(* CODESYS project CtaAppLeistungsventile_2.0.0.0.library
   Description: Leistungventile Library der CTA
   Version: 2.0.0.0
   Title: CtaAppLeistungventile
   Author: SIS
   DocFormat: reStructuredText
   Placeholder: CtaAppLeistungventile
   LanguageModelAttribute: qualified-access-only
   DefaultNamespace: CtaAppLeistungventile
   CompiledLibraryCompatibilityVersion: CODESYS V3.5 SP16 Patch 3
   Company: CTA

Project tree, tasks and I/O mapping:
  libraries: Standard, 3.5.18.0 (System); CtaSysConfig, 2.0.0.0 (CTA); VisuDialogs, 3.5.16.20 (System); VisuSymbols, 4.5.0.0 (System); CtaVisSymbols, 2.0.0.0 (CTA); CtaAppInfluxLog, 1.0.0.1 (CTA); CtaSysIO, 2.0.0.0 (CTA); CtaSysLeistungventile, 2.0.0.0 (CTA); CtaVisApps, 1.0.0.0 (CTA); CtaVisHelp, 2.0.0.0 (CTA); CtaVisUser, 1.0.0.0 (CTA)
  40 Visualizations/
    CSH/
      PARAMETER/
        visualisation VIS_CSH_PARAMETER
      VISU/
        visualisation VIS_CSH
        visualisation VIS_CSH_QUERY
      ITF_PARAMETER/
        visualisation DIA_CSH_PARAMETER_IO_ITF
      visualisation DIA_CSH
  00000000-0000-0000-0000-000000000000|D:\CoDeSys\LibrariesV3\trunk\Intern\CAA\CAA Template\3.4.0.0 draft\Placeholder.xml
  00000000-0000-0000-0000-000000000000|D:\CoDeSys\LibrariesV3\trunk\Intern\CAA\CAA Template\3.2.0.3 draft\Prefix.pdf
  00000000-0000-0000-0000-000000000000|D:\CoDeSys\LibrariesV3\trunk\Intern\CAA\CAA Template\3.5.2.0 draft\Placeholder.xml
  20 Structs/
    CSV/
      data type scParameter
  50 Images/
  10 Documenation/
    global variables VersionHistory
    global variables readMe
  21 Interface/
    interface ITF_CSH: pro_ITF_CR2, pro_ITF_CR3, pro_ITF_CR4, pro_ITF_CR1, P_tTillCAPStart, P_tTillCAP25, P_tTillCAP100, P_tCR4OffOn
  11 Library Parameter/
  12 Konstanten/
  60 Textlisten/
  13 Globale Variablen/
  text list GlobalTextList
  5ce3da45-db07-42e7-a21c-a00fff4ed8f6|C:\Users\sis\Downloads\dip-switch.svg
  5ce3da45-db07-42e7-a21c-a00fff4ed8f6|C:\Users\sis\Downloads\lightning-bolt-circle.svg
  30 Program Organization Units/
    function block FB_CSH [ST]: metDO_CR4_ON, proDO_CR4_ON, proCR4_ON_ITF, pro_ITF_CR1, pro_ITF_CR2, pro_ITF_CR3, pro_ITF_CR4, actConfig, actTrendLog, P_tCR4OffOn, P_tTillCAP100, P_tTillCAP25, P_tTillCAPStart, metDO_CR1_ON, proDO_CR1_ON, proCR1_ON_ITF, metDO_CR2_ON, proDO_CR2_ON, proCR2_ON_ITF, metDO_CR3_ON, proDO_CR3_ON, proCR3_ON_ITF, FB_INIT
  5ce3da45-db07-42e7-a21c-a00fff4ed8f6|C:\Users\sis\Downloads\sine-wave.svg
  5ce3da45-db07-42e7-a21c-a00fff4ed8f6|C:\Users\sis\Downloads\eye.svg
  5ce3da45-db07-42e7-a21c-a00fff4ed8f6|C:\Users\sis\Downloads\lan.svg
*)

// 20 Structs/CSV/scParameter
TYPE scParameter :
	STRUCT
		tTillCAPStart	:	CtaSysConfig.fbTIME;
		tTillCAP25		:	CtaSysConfig.fbTIME;
		tTillCAP100		:	CtaSysConfig.fbTIME;	
		tCR4OffOn		:	CtaSysConfig.fbTIME;		
	END_STRUCT
END_TYPE

// 10 Documenation/VersionHistory
(* 

.. image:: ../../Images/CTA_Logo.jpg
   :align: right
   :width: 15% 

**Vorlage**   


============ =========== =========== ============================================
**Date**     **Version** **Author**  **Change**
------------ ----------- ----------- --------------------------------------------
04.03.2021   0.0.0.0     SIS         Vorlage erstellt

============ =========== =========== ============================================


*)
VAR_GLOBAL
    stInfo : STRING:= '0.0.0.0, Vorlage, CTA';
END_VAR

// 10 Documenation/readMe
(*

**ReadMe**
 
|	**Empfehlung**
|
|	Bibliothek CtaAppFU zur dämpfung und rampung von Signalen
|	Instanzieren Sie den CtaAppFU.fbFU in ihrem Funktionsbaustein oder POU beispielsweise als fbFUx ( x = Nr. des FU's 
|	Deklarieren Sie die Struktur Variable welche als Parameter und zur ansteuerung dienen wie im Code beispiel.
|  
| *Beispiel* 

+-----------------------+---------------------------------------------------------------------------------------------------------------------------------------------------------------------------------------------------------------------------------------------------------------------------------------------------------------------------------------------------------------------------------------------------------------------------------------+
| Beschreibung          |  Code                                                                                                                                                                                                                                                                                                                                                                                                                                 |
+=======================+=======================================================================================================================================================================================================================================================================================================================================================================================================================================+
| POU oder SmFb         | .. code-block:: codesys                                                                                                                                                                                                                                                                                                                                                                                                               |
|                       |                                                                                                                                                                                                                                                                                                                                                                                                                                       |
|                       |	// Deklaration als VAR im POU oder dem selbsterstellten Funktionsbaustein                                                                                                                                                                                                                                                                                                                                                        	|
|                       |   VAR   																																																				 																																																				|
|						|	    (*Frequenzumformer 1*)																																																		 																																																	|
|						|		fbFU1			: CtaAppFU.fbFU;																																																																																																|
|			 			|	END_VAR                                                                                                                                                                                                                                                                                                                                                                                                                          	|
+-----------------------+---------------------------------------------------------------------------------------------------------------------------------------------------------------------------------------------------------------------------------------------------------------------------------------------------------------------------------------------------------------------------------------------------------------------------------------+
| Code für Init         | .. code-block:: codesys                                                                                                                                                                                                                                                                                                                                                                                                               |
|                       |   																																																					 																																																				|
|			 			|	// Kopieren des nachfolgenden Codes in eine Action zur Initialisierung der Parameter. Zum Beispiel actConfig.																																																				 																										|
|                       |	{region "Parameter Temperaturfühler 1"}                                                                                                                                                                                                                                                                                                                                                                                             |
|			 			|		(*Basis*)                                                                                                                                                                                                                                                                                                                                                                                                                       |
|						|		fbFU1.scParameter.scModBus.fbxMbErrorAsWarning					(_WertInit := FALSE																	 	 		);     //P1 Parameter zur behandlung eines ModBus Fehlers als Warnung.																																															|
|						|	{endregion}                                                                                                                                                      																																																																    | 
|						|																																																																																																										|
+-----------------------+---------------------------------------------------------------------------------------------------------------------------------------------------------------------------------------------------------------------------------------------------------------------------------------------------------------------------------------------------------------------------------------------------------------------------------------+
*)                                                                                                                                                                                                                                                                                                                                                                                                                                                               
VAR_GLOBAL
	xReadMeDone              :   BOOL; 
END_VAR

// 30 Program Organization Units/FB_CSH
FUNCTION_BLOCK FB_CSH EXTENDS CtaSysLeistungventile.FB_LEISTUNGSVENTILE_BASE IMPLEMENTS ITF_CSH
VAR_INPUT
END_VAR
VAR_OUTPUT
END_VAR
VAR	
	// TON
	TON_CAPStart		:	Standard.TON;
	TON_CR4On			:	Standard.TON;	
	TON_CR4Off			:	Standard.TON;
	TON_CAPUp			:	Standard.TON;
	TON_CAPDown			:	Standard.TON;

	// CASE VARIABLEN
	iStepCAPUP			:	INT	:= 1;
	iStepCAPDown		:	INT	:= 1;
	
	// FLANKEN
	pUp					:	Standard.R_TRIG;
	pDown				:	Standard.R_TRIG;
	
	// ZU UND WEGSCHALTZEITEN
	tPerCAPUp			:	TIME;
	tPerCAPDown			:	TIME;
	
	(* Trend Log *)
	fbTrendxCr1			:	CtaAppInfluxLog.FB_LOG_NODE_BOOL;
	fbTrendxCr2			:	CtaAppInfluxLog.FB_LOG_NODE_BOOL;
	fbTrendxCr3			:	CtaAppInfluxLog.FB_LOG_NODE_BOOL;
	fbTrendxCr4			:	CtaAppInfluxLog.FB_LOG_NODE_BOOL;
	fbTrendiCap			:	CtaAppInfluxLog.FB_LOG_NODE_INT;
	
	// Var
	
	xHasBeenReleasedFirst	:	BOOL;
	(* Config *)
	fbConfigFile		:	CtaSysConfig.fbConfigFile;	
	scParameter			:	scParameter;
END_VAR

actConfig();

tPerCAPUp 	:=	scParameter.tTillCAP100.proValue 	/ 4;
tPerCAPDown :=	scParameter.tTillCAP25.proValue		/ 4;	

// Generation of pulses for CR4
TON_CR4On(In := NOT TON_CR4Off.Q ,PT := scParameter.tCR4OffOn.proValue);
TON_CR4Off(In := TON_CR4On.Q ,PT := scParameter.tCR4OffOn.proValue);

IF proRelease THEN
	
	iStepCAPDown := 1;
	
	TON_CAPStart(In := proRelease ,PT := scParameter.tTillCAPStart.proValue);
	
	xHasBeenReleasedFirst := TRUE;
	
	IF TON_CAPStart.Q THEN
		IF scParameter.tTillCAP100.proValue <= T#0S THEN	
			xCR1	:= FALSE;
			xCR2	:= FALSE;
			xCR3 	:= FALSE;
			xCR4	:= TON_CR4On.Q;
			
			xAcknowledge := FALSE;	
		ELSE
			
			xAcknowledge := TRUE;
			
			pUp(CLK := TON_CAPUp.Q);
		
			IF pUp.Q AND iStepCAPUP >= 1 AND iStepCAPUP < 4 THEN
				iStepCAPUP := iStepCAPUP + 1;
			END_IF
	
			CASE iStepCAPUP OF				
			
				1:	// 25%
					xCR1 := FALSE;
					xCR2 := FALSE;
					xCR3 := TRUE;
					xCR4 :=  TON_CR4On.Q;
					iCAP := 25;
			
				2:	// 50%
					xCR1 := FALSE;
					xCR2 := TRUE;
					xCR3 := FALSE;
					xCR4 := TON_CR4On.Q;
					iCAP := 50;
					
				3:	// 75%
					xCR1 := TRUE;
					xCR2 := FALSE;
					xCR3 := FALSE;
					xCR4 := TON_CR4On.Q;
					iCAP := 75;
					
				4:	// 100%
					xCR1 := FALSE;
					xCR2 := FALSE;
					xCR3 := FALSE;
					xCR4 := TON_CR4On.Q;
					iCAP := 100;			
			END_CASE
			
			TON_CAPUp(	IN := NOT TON_CAPUp.Q AND iStepCAPUP < 4,
							PT := tPerCAPUp);
			
		END_IF			
	
	ELSE
		xCR1 := FALSE;
		xCR2 := FALSE;
		xCR3 := TRUE;
		xCR4 := FALSE;
		
		xAcknowledge := FALSE;
	END_IF
ELSE
	IF xHasBeenReleasedFirst THEN
		
		iStepCAPUP := 1;
		
		pDown(CLK := TON_CAPDown.Q);
	
		IF pDown.Q AND iStepCAPDown >= 1 AND iStepCAPDown < 4 THEN
			iStepCAPDown := iStepCAPDown + 1;
		END_IF		
		
		CASE iStepCAPDown OF		
			
				1: // 75%
					xCR1 := TRUE;
					xCR2 := FALSE;
					xCR3 := FALSE;
					xCR4 := TON_CR4On.Q;
					iCAP := 75;
					xAcknowledge := TRUE;
				2: // 50%
					xCR1 := FALSE;
					xCR2 := TRUE;
					xCR3 := FALSE;
					xCR4 := TON_CR4On.Q;
					iCAP := 50;
					xAcknowledge := TRUE;
				3: // 25%
					xCR1 := FALSE;
					xCR2 := FALSE;
					xCR3 := TRUE;
					xCR4 :=  TON_CR4On.Q;
					iCAP := 25;
					xAcknowledge := TRUE;
				4: // Stop
					xCR1 := FALSE;
					xCR2 := FALSE;
					xCR3 := TRUE;
					xCR4 := FALSE;	
					iCAP := 25;
					xAcknowledge := FALSE;	
					xHasBeenReleasedFirst := FALSE;
		END_CASE	
		
		TON_CAPDown(	IN := NOT TON_CAPDown.Q AND iStepCAPDown < 4,
						PT := tPerCAPDown);
	END_IF	
END_IF

IF __QUERYINTERFACE(ITF_BMK,ITF_BMK) THEN
	actTrendlog();
END_IF

METHOD metDO_CR4_ON : BOOL
VAR_INPUT
    ITF_IN		:	CtaSysIO.ITF_IO;
END_VAR
VAR	
	ITF_DO		:	CtaSysIO.ITF_DO;
END_VAR
IF ITF_IN <> 0 THEN	
	ITF_xCR4_ON := ITF_IN;
	IF __QUERYINTERFACE(ITF_xCR4_ON,ITF_DO) THEN		
		ITF_DO.proValue := xCR4;
	END_IF	
ELSE
	metDO_CR4_ON := xCR4;
END_IF
END_METHOD

PROPERTY proDO_CR4_ON : BOOL
GET
proDO_CR4_ON := xCR4;
END_GET
END_PROPERTY

PROPERTY proCR4_ON_ITF : CtaSysIO.ITF_IO
GET
proCR4_ON_ITF := ITF_xCR4_ON;
END_GET
END_PROPERTY

PROPERTY pro_ITF_CR1 : CtaSysIO.ITF_IO
GET
pro_ITF_CR1 := ITF_xCR1_ON;
END_GET
END_PROPERTY

PROPERTY pro_ITF_CR2 : CtaSysIO.ITF_IO
GET
pro_ITF_CR2 := ITF_xCR2_ON;
END_GET
END_PROPERTY

PROPERTY pro_ITF_CR3 : CtaSysIO.ITF_IO
GET
pro_ITF_CR3 := ITF_xCR3_ON;
END_GET
END_PROPERTY

PROPERTY pro_ITF_CR4 : CtaSysIO.ITF_IO
GET
pro_ITF_CR4 := ITF_xCR4_ON;
END_GET
END_PROPERTY

ACTION actConfig:
fbConfigFile();

	scParameter.tTillCAPStart	(_usiParaNr := 1,	itfConfigFb := fbConfigFile);
	scParameter.tTillCAP25		(_usiParaNr := 2,	itfConfigFb := fbConfigFile);
	scParameter.tTillCAP100		(_usiParaNr := 3,	itfConfigFb := fbConfigFile);
	scParameter.tCR4OffOn		(_usiParaNr := 4,	itfConfigFb := fbConfigFile);
END_ACTION

ACTION actTrendLog:
(* CR1 *)
fbTrendxCr1.ENABLE		:= TRUE;
fbTrendxCr1.KEY			:= CONCAT(ITF_BMK.proGetObjectId,'_xCR1');
fbTrendxCr1.SET_VALUE	:= xCR1;

(* CR2 *)
fbTrendxCr2.ENABLE		:= TRUE;
fbTrendxCr2.KEY			:= CONCAT(ITF_BMK.proGetObjectId,'_xCR2');
fbTrendxCr2.SET_VALUE	:= xCR2;

(* CR3 *)
fbTrendxCr3.ENABLE		:= TRUE;
fbTrendxCr3.KEY			:= CONCAT(ITF_BMK.proGetObjectId,'_xCR3');
fbTrendxCr3.SET_VALUE	:= xCR3;

(* CR4 *)
fbTrendxCr4.ENABLE		:= TRUE;
fbTrendxCr4.KEY			:= CONCAT(ITF_BMK.proGetObjectId,'_xCR4');
fbTrendxCr4.SET_VALUE	:= xCR4;

(* actCAP *)
fbTrendiCap.ENABLE		:= TRUE;
fbTrendiCap.KEY			:= CONCAT(ITF_BMK.proGetObjectId,'_iCAP');
fbTrendiCap.SET_VALUE	:= iCAP;
END_ACTION

PROPERTY P_tCR4OffOn : CtaSysConfig.ITF_DATATYPE
GET
P_tCR4OffOn := scParameter.tCR4OffOn;
END_GET
END_PROPERTY

PROPERTY P_tTillCAP100 : CtaSysConfig.ITF_DATATYPE
GET
P_tTillCAP100 := scParameter.tTillCAP100;
END_GET
END_PROPERTY

PROPERTY P_tTillCAP25 : CtaSysConfig.ITF_DATATYPE
GET
P_tTillCAP25 := scParameter.tTillCAP25;
END_GET
END_PROPERTY

PROPERTY P_tTillCAPStart : CtaSysConfig.ITF_DATATYPE
GET
P_tTillCAPStart := scParameter.tTillCAPStart;
END_GET
END_PROPERTY

METHOD metDO_CR1_ON : BOOL
VAR_INPUT
    ITF_IN		:	CtaSysIO.ITF_IO;
END_VAR
VAR	
	ITF_DO		:	CtaSysIO.ITF_DO;
END_VAR
IF ITF_IN <> 0 THEN	
	ITF_xCR1_ON := ITF_IN;
	IF __QUERYINTERFACE(ITF_xCR1_ON,ITF_DO) THEN		
		ITF_DO.proValue := xCR1;
	END_IF	
ELSE
	metDO_CR1_ON := xCR1;
END_IF
END_METHOD

PROPERTY proDO_CR1_ON : BOOL
GET
proDO_CR1_ON := xCR1;
END_GET
END_PROPERTY

PROPERTY proCR1_ON_ITF : CtaSysIO.ITF_IO
GET
proCR1_ON_ITF := ITF_xCR1_ON;
END_GET
END_PROPERTY

METHOD metDO_CR2_ON : BOOL
VAR_INPUT
    ITF_IN		:	CtaSysIO.ITF_IO;
END_VAR
VAR	
	ITF_DO		:	CtaSysIO.ITF_DO;
END_VAR
IF ITF_IN <> 0 THEN	
	ITF_xCR2_ON := ITF_IN;
	IF __QUERYINTERFACE(ITF_xCR2_ON,ITF_DO) THEN		
		ITF_DO.proValue := xCR2;
	END_IF	
ELSE
	metDO_CR2_ON := xCR2;
END_IF
END_METHOD

PROPERTY proDO_CR2_ON : BOOL
GET
proDO_CR2_ON := xCR2;
END_GET
END_PROPERTY

PROPERTY proCR2_ON_ITF : CtaSysIO.ITF_IO
GET
proCR2_ON_ITF := ITF_xCR2_ON;
END_GET
END_PROPERTY

METHOD metDO_CR3_ON : BOOL
VAR_INPUT
    ITF_IN		:	CtaSysIO.ITF_IO;
END_VAR
VAR	
	ITF_DO		:	CtaSysIO.ITF_DO;
END_VAR
IF ITF_IN <> 0 THEN	
	ITF_xCR3_ON := ITF_IN;
	IF __QUERYINTERFACE(ITF_xCR3_ON,ITF_DO) THEN		
		ITF_DO.proValue := xCR3;
	END_IF	
ELSE
	metDO_CR3_ON := xCR3;
END_IF
END_METHOD

PROPERTY proDO_CR3_ON : BOOL
GET
proDO_CR3_ON := xCR3;
END_GET
END_PROPERTY

PROPERTY proCR3_ON_ITF : CtaSysIO.ITF_IO
GET
proCR3_ON_ITF := ITF_xCR3_ON;
END_GET
END_PROPERTY

//FB_Init ist immer implizit verfügbar und wird primär für die Initialisierung verwendet.
//Der Rückgabewert wird nicht ausgewertet. Für gezielte Einflussnahme können Sie
//die Methoden explizit deklarieren und darin mit dem Standard-Initialisierungscode 
//zusätzlichen Code bereitstellen. Sie können den Rückgabewert auswerten.
METHOD FB_Init: BOOL
VAR_INPUT    
bInitRetains: BOOL; // TRUE: Die Retain-Variablen werden initialisiert (Reset warm / Reset kalt)    
bInCopyCode: BOOL;  // TRUE: Die Instanz wird danach in den Kopiercode kopiert (Online-Change)
END_VAR
SUPER^.stVisuDiaName := 'CtaAppLeistungventile.DIA_CSH';
END_METHOD

END_FUNCTION_BLOCK

// 21 Interface/ITF_CSH
INTERFACE ITF_CSH EXTENDS CtaSysLeistungventile.ITF_LEISTUNGSVENTILE_BASE

PROPERTY pro_ITF_CR2 : CtaSysIO.ITF_IO
GET
END_GET
END_PROPERTY

PROPERTY pro_ITF_CR3 : CtaSysIO.ITF_IO
GET
END_GET
END_PROPERTY

PROPERTY pro_ITF_CR4 : CtaSysIO.ITF_IO
GET
END_GET
END_PROPERTY

PROPERTY pro_ITF_CR1 : CtaSysIO.ITF_IO
GET
END_GET
END_PROPERTY

PROPERTY P_tTillCAPStart : CtaSysConfig.ITF_DATATYPE
GET
END_GET
END_PROPERTY

PROPERTY P_tTillCAP25 : CtaSysConfig.ITF_DATATYPE
GET
END_GET
END_PROPERTY

PROPERTY P_tTillCAP100 : CtaSysConfig.ITF_DATATYPE
GET
END_GET
END_PROPERTY

PROPERTY P_tCR4OffOn : CtaSysConfig.ITF_DATATYPE
GET
END_GET
END_PROPERTY

END_INTERFACE

// 40 Visualizations/CSH/PARAMETER/VIS_CSH_PARAMETER
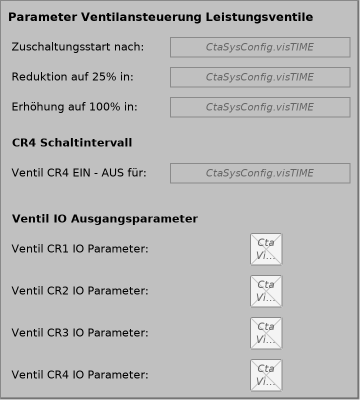
VISUALIZATION VIS_CSH_PARAMETER  // 360x400
VAR_INPUT	
	ITF_CSH_IN				:	ITF_CSH;
	ITF_CR1_IN				:	CtaSysIO.ITF_IO;
	ITF_CR2_IN				:	CtaSysIO.ITF_IO;
	ITF_CR3_IN				:	CtaSysIO.ITF_IO;
	ITF_CR4_IN				:	CtaSysIO.ITF_IO;	
END_VAR
    RoundedRectangle (0,0 358x398)
    Frame (170,37 180x20)
        shows CtaSysConfig.visTIME(visfbTIMEIn := ITF_CSH_IN.P_tTillCAPStart)
    Frame (170,67 180x20)
        shows CtaSysConfig.visTIME(visfbTIMEIn := ITF_CSH_IN.P_tTillCAP25)
    Frame (170,97 180x20)
        shows CtaSysConfig.visTIME(visfbTIMEIn := ITF_CSH_IN.P_tTillCAP100)
    Frame (170,163 180x20)
        shows CtaSysConfig.visTIME(visfbTIMEIn := ITF_CSH_IN.P_tCR4OffOn)
    Label (5,37 150x20), "Zuschaltungsstart nach:"
    Label (5,67 150x20), "Reduktion auf 25% in:"
    Label (5,97 150x20), "Erhöhung auf 100% in:"
    Label (5,163 150x20), "Ventil CR4 EIN - AUS für:"
    Label (5,233 150x32), "Ventil CR1 IO Parameter:", invisible if: ITF_CR1_IN = 0
    Label (5,275 150x32), "Ventil CR2 IO Parameter:", invisible if: ITF_CR2_IN = 0
    Label (5,317 150x32), "Ventil CR3 IO Parameter:", invisible if: ITF_CR3_IN = 0
    Label (5,359 150x32), "Ventil CR4 IO Parameter:", invisible if: ITF_CR4_IN = 0
    Image (250,233 32x32), invisible if: ITF_CR1_IN = 0, input disabled if: ITF_CR1_IN = 0, image: CtaVisSymbols.ImagePool.build
        OnMouseClick:  Dialog=DIA_CSH_PARAMETER_IO_ITF, Parameters={ITF_IO_IN: ITF_CR1_IN}, OpenModal=True, OpenCentered=True
    Image (250,275 32x32), invisible if: ITF_CR2_IN = 0, input disabled if: ITF_CR2_IN = 0, image: CtaVisSymbols.ImagePool.build
        OnMouseClick:  Dialog=DIA_CSH_PARAMETER_IO_ITF, Parameters={ITF_IO_IN: ITF_CR2_IN}, OpenModal=True, OpenCentered=True
    Image (250,317 32x32), invisible if: ITF_CR3_IN = 0, input disabled if: ITF_CR3_IN = 0, image: CtaVisSymbols.ImagePool.build
        OnMouseClick:  Dialog=DIA_CSH_PARAMETER_IO_ITF, Parameters={ITF_IO_IN: ITF_CR3_IN}, OpenModal=True, OpenCentered=True
    Image (250,359 32x32), invisible if: ITF_CR4_IN = 0, input disabled if: ITF_CR4_IN = 0, image: CtaVisSymbols.ImagePool.build
        OnMouseClick:  Dialog=DIA_CSH_PARAMETER_IO_ITF, Parameters={ITF_IO_IN: ITF_CR4_IN}, OpenModal=True, OpenCentered=True
    Label (5,133 250x20), "CR4 Schaltintervall"
    Label (5,7 350x20), "Parameter Ventilansteuerung Leistungsventile"
    Label (5,209 250x20), "Ventil IO Ausgangsparameter", invisible if: ITF_CR1_IN = 0 AND ITF_CR2_IN = 0 AND ITF_CR3_IN = 0 AND ITF_CR4_IN = 0
END_VISUALIZATION

// 40 Visualizations/CSH/VISU/VIS_CSH
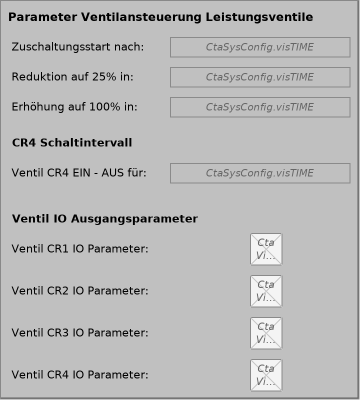
VISUALIZATION VIS_CSH  // 360x400
VAR_INPUT
	ITF_CSH_IN	:	ITF_CSH;
END_VAR
    Frame (0,0 360x400), invisible if: NOT __QUERYINTERFACE(ITF_CSH_IN,ITF_CSH_IN)
        shows VIS_CSH_QUERY(ITF_CSH_IN := ITF_CSH_IN)
END_VISUALIZATION

// 40 Visualizations/CSH/VISU/VIS_CSH_QUERY
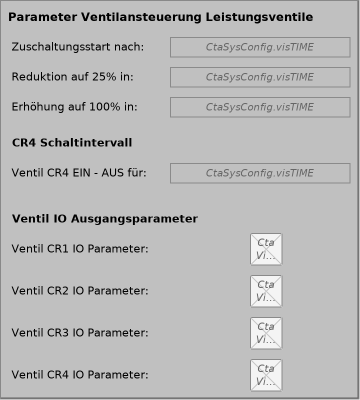
VISUALIZATION VIS_CSH_QUERY  // 360x400
VAR_INPUT
	ITF_CSH_IN	:	ITF_CSH;
END_VAR
    Frame (0,0 360x400)
        shows VIS_CSH_PARAMETER(ITF_CSH_IN := ITF_CSH_IN, ITF_CR1_IN := ITF_CSH_IN.pro_ITF_CR1, ITF_CR2_IN := ITF_CSH_IN.pro_ITF_CR2, ITF_CR3_IN := ITF_CSH_IN.pro_ITF_CR3, ITF_CR4_IN := ITF_CSH_IN.pro_ITF_CR4)
END_VISUALIZATION

// 40 Visualizations/CSH/ITF_PARAMETER/DIA_CSH_PARAMETER_IO_ITF
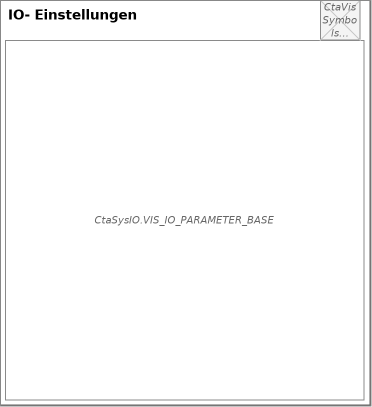
VISUALIZATION DIA_CSH_PARAMETER_IO_ITF  // 372x407
VAR_INPUT
    ITF_IO_IN    :   CtaSysIO.ITF_IO;	
END_VAR
    RoundedRectangle (0,0 370x405)
    Frame (5,40 359x360)
        shows CtaSysIO.VIS_IO_PARAMETER_BASE(ITF_IO_IN := ITF_IO_IN)
        shows VIS_ANTRIEB_PARAMETER_IO1(ITF_ANTRIEBIN := ITF_ANTRIEBIN)
        shows VIS_ANTRIEB_PARAMETER_IO2(ITF_ANTRIEBIN := ITF_ANTRIEBIN)
        shows VIS_ANTRIEB_PARAMETER_IO3(ITF_ANTRIEBIN := ITF_ANTRIEBIN)
    Image (320,0 40x40), image: CtaVisSymbols.ImagePool.close_solo_black
        OnMouseClick:  Dialog=DIA_CSH_PARAMETER_IO_ITF, Result=None, NumpadKeypadSet=True
    Label (5,5 150x20), "IO- Einstellungen"
END_VISUALIZATION

// 40 Visualizations/CSH/DIA_CSH
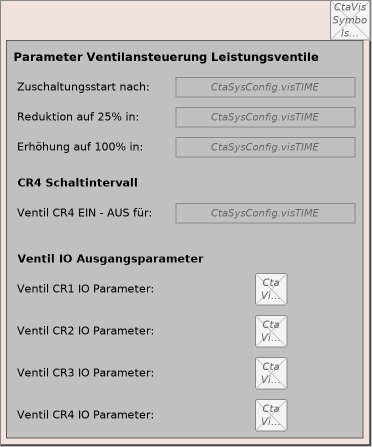
VISUALIZATION DIA_CSH  // 372x447
VAR_INPUT
	ITF_CSH_BASE_IN 	:	CtaSysLeistungventile.ITF_LEISTUNGSVENTILE_BASE;
END_VAR
VAR
	ITF_CSH_QUERRY		:	ITF_CSH;
END_VAR
    RoundedRectangle (0,0 370x445)
    Image (330,0 40x40), image: CtaVisSymbols.ImagePool.close_solo_black
        OnMouseClick:  Dialog=DIA_CSH, Result=OK, NumpadKeypadSet=True
    Frame (6,40 359x400), invisible if: NOT __QUERYINTERFACE(ITF_CSH_BASE_IN,ITF_CSH_QUERRY)
        shows VIS_CSH(ITF_CSH_IN := ITF_CSH_QUERRY)
END_VISUALIZATION
